{attribute 'qualified_only'}
{attribute 'strict'}
{attribute 'to_string'}
TYPE E_Example :
(
	red := -1,
	blue,
	green
) SINT := blue; //Definfes this as a SINT with a default value of blue
END_TYPE

(* stored: Version 1.1.0.1
   DUT E_Example: Id {2d3ab809-9480-4556-ada3-70e7f2983408} *)
